FUNCTION_BLOCK IA_COGSOGRapidUpdate (* ISOBUS Adapter for Course Over Ground and Speed Over Ground (Rapid Update) *)
  (* Standard: NMEA 2000; Classification: PGN 129026; Description: Copyright (c) 2024-2026 HR Agrartechnik GmbH This program and the accompanying materials are made available under the terms of the Eclipse Public License 2.0 which is available at https://www.eclipse.org/legal/epl-2.0/ SPDX-License-Identifier: EPL-2.0 *)
  (* Version 1.0, 2026-04-19, Franz Höpfinger, HR Agrartechnik GmbH, initial API and implementation (Adapter Wrapper for I_COGSOGRapidUpdate) *)
  PACKAGE isobus::tecu;
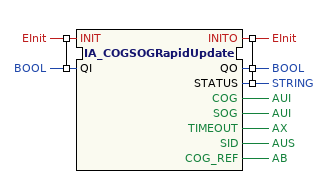
  EVENT_INPUT
    INIT : EInit WITH QI; (* Service Initialization *)
  END_EVENT
  EVENT_OUTPUT
    INITO : EInit WITH QO, STATUS; (* Initialization Confirm *)
  END_EVENT
  VAR_INPUT
    QI : BOOL; (* Event Input Qualifier *)
  END_VAR
  VAR_OUTPUT
    QO : BOOL; (* Event Output Qualifier *)
    STATUS : STRING;
  END_VAR
  PLUGS
    COG : adapter::types::unidirectional::AUI; (* Course Over Ground *)
    SOG : adapter::types::unidirectional::AUI; (* Speed Over Ground *)
    TIMEOUT : adapter::types::unidirectional::AX; (* Timeout Status *)
    SID : adapter::types::unidirectional::AUS; (* Sequence ID *)
    COG_REF : adapter::types::unidirectional::AB; (* COG Reference *)
  END_PLUGS
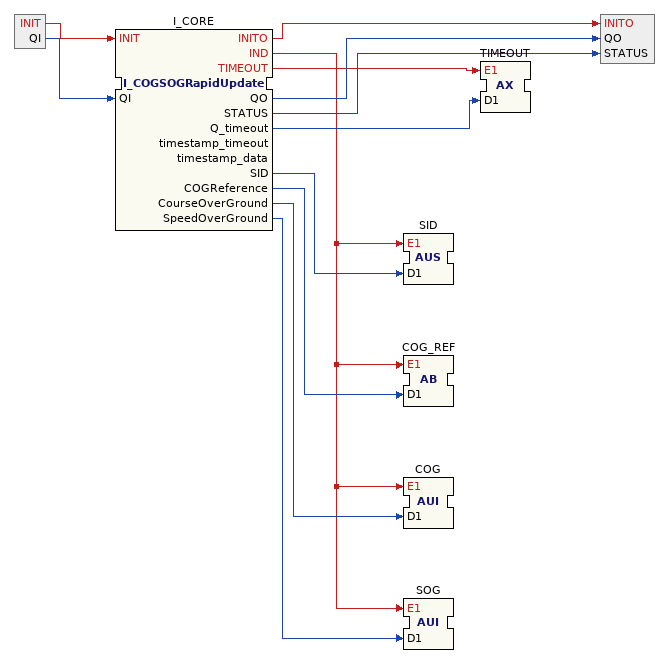
  FBS
    I_CORE : isobus::tecu::I_COGSOGRapidUpdate;
  END_FBS
  EVENT_CONNECTIONS
    INIT TO I_CORE.INIT;
    I_CORE.INITO TO INITO;
    I_CORE.IND TO COG.E1;
    I_CORE.IND TO SOG.E1;
    I_CORE.IND TO SID.E1;
    I_CORE.IND TO COG_REF.E1;
    I_CORE.TIMEOUT TO TIMEOUT.E1;
  END_CONNECTIONS
  DATA_CONNECTIONS
    QI TO I_CORE.QI;
    I_CORE.QO TO QO;
    I_CORE.STATUS TO STATUS;
    I_CORE.CourseOverGround TO COG.D1;
    I_CORE.SpeedOverGround TO SOG.D1;
    I_CORE.Q_timeout TO TIMEOUT.D1;
    I_CORE.SID TO SID.D1;
    I_CORE.COGReference TO COG_REF.D1;
  END_CONNECTIONS
END_FUNCTION_BLOCK
